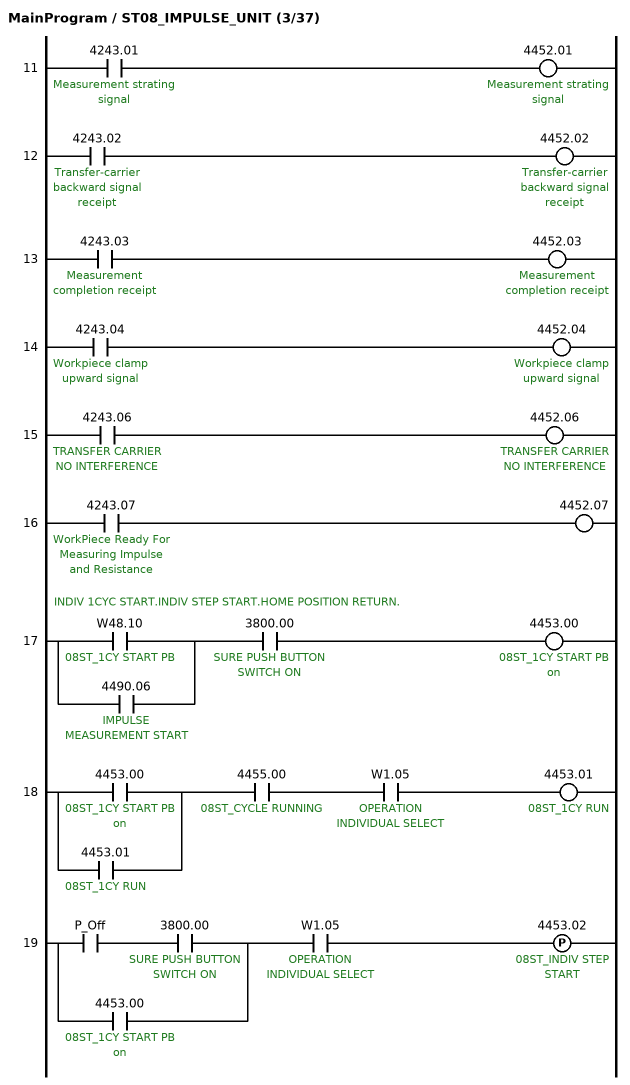
; [picture p432: MainProgram / ST08_IMPULSE_UNIT, rungs 11-19]
; rung 11
LD 4243.01  ; Measurement strating signal
OUT 4452.01  ; Measurement strating signal
; rung 12
LD 4243.02  ; Transfer-carrier backward signal receipt
OUT 4452.02  ; Transfer-carrier backward signal receipt
; rung 13
LD 4243.03  ; Measurement completion receipt
OUT 4452.03  ; Measurement completion receipt
; rung 14
LD 4243.04  ; Workpiece clamp upward signal
OUT 4452.04  ; Workpiece clamp upward signal
; rung 15
LD 4243.06  ; TRANSFER CARRIER NO INTERFERENCE
OUT 4452.06  ; TRANSFER CARRIER NO INTERFERENCE
; rung 16
LD 4243.07  ; WorkPiece Ready For Measuring Impulse and Resistance
OUT 4452.07
; rung 17: INDIV 1CYC START.INDIV STEP START.HOME POSITION RETURN.
LD W48.10  ; 08ST_1CY START PB
OR 4490.06  ; IMPULSE MEASUREMENT START
AND 3800.00  ; SURE PUSH BUTTON SWITCH ON
OUT 4453.00  ; 08ST_1CY START PB on
; rung 18
LD 4453.00  ; 08ST_1CY START PB on
OR 4453.01  ; 08ST_1CY RUN
AND 4455.00  ; 08ST_CYCLE RUNNING
AND W1.05  ; OPERATION INDIVIDUAL SELECT
OUT 4453.01  ; 08ST_1CY RUN
; rung 19
LD P_Off
AND 3800.00  ; SURE PUSH BUTTON SWITCH ON
OR 4453.00  ; 08ST_1CY START PB on
AND W1.05  ; OPERATION INDIVIDUAL SELECT
DIFU(013) 4453.02  ; 08ST_INDIV STEP START

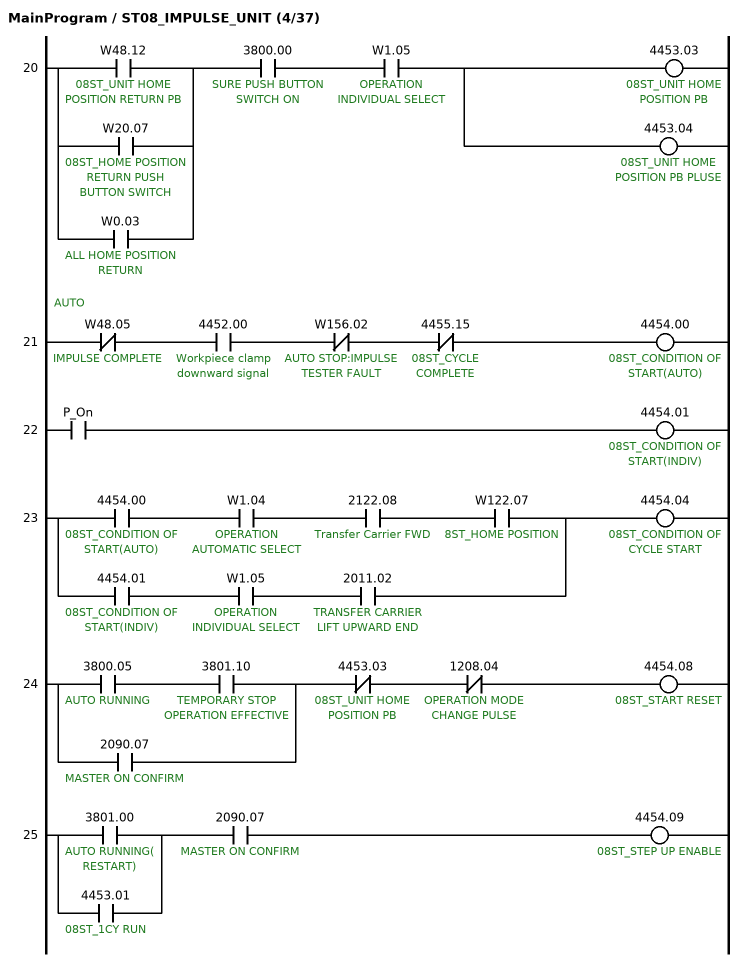
; rung 20
LD W48.12  ; 08ST_UNIT HOME POSITION RETURN PB
OR W20.07  ; 08ST_HOME POSITION RETURN PUSH BUTTON SWITCH
OR W0.03  ; ALL HOME POSITION RETURN
AND 3800.00  ; SURE PUSH BUTTON SWITCH ON
AND W1.05  ; OPERATION INDIVIDUAL SELECT
OUT 4453.03  ; 08ST_UNIT HOME POSITION PB
OUT 4453.04  ; 08ST_UNIT HOME POSITION PB PLUSE
; rung 21: AUTO
LDNOT W48.05  ; IMPULSE COMPLETE
AND 4452.00  ; Workpiece clamp downward signal
ANDNOT W156.02  ; AUTO STOP:IMPULSE TESTER FAULT
ANDNOT 4455.15  ; 08ST_CYCLE COMPLETE
OUT 4454.00  ; 08ST_CONDITION OF START(AUTO)
; rung 22
LD P_On
OUT 4454.01  ; 08ST_CONDITION OF START(INDIV)
; rung 23
LD 4454.00  ; 08ST_CONDITION OF START(AUTO)
AND W1.04  ; OPERATION AUTOMATIC SELECT
AND 2122.08  ; Transfer Carrier FWD
AND W122.07  ; 8ST_HOME POSITION
LD 4454.01  ; 08ST_CONDITION OF START(INDIV)
AND W1.05  ; OPERATION INDIVIDUAL SELECT
AND 2011.02  ; TRANSFER CARRIER LIFT UPWARD END
ORLD
OUT 4454.04  ; 08ST_CONDITION OF CYCLE START
; rung 24
LD 3800.05  ; AUTO RUNNING
AND 3801.10  ; TEMPORARY STOP OPERATION EFFECTIVE
OR 2090.07  ; MASTER ON CONFIRM
ANDNOT 4453.03  ; 08ST_UNIT HOME POSITION PB
ANDNOT 1208.04  ; OPERATION MODE CHANGE PULSE
OUT 4454.08  ; 08ST_START RESET
; rung 25
LD 3801.00  ; AUTO RUNNING(RESTART)
OR 4453.01  ; 08ST_1CY RUN
AND 2090.07  ; MASTER ON CONFIRM
OUT 4454.09  ; 08ST_STEP UP ENABLE

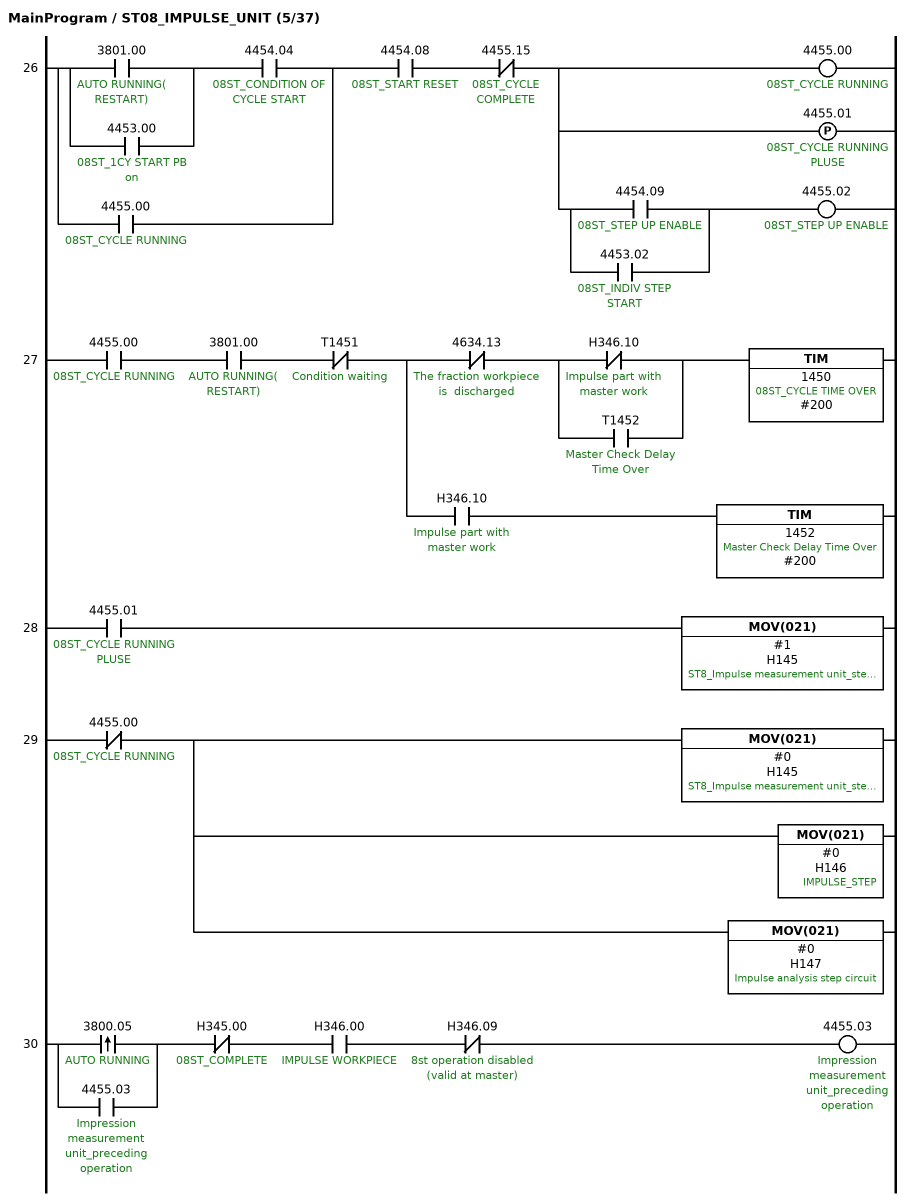
; rung 26
LD 3801.00  ; AUTO RUNNING(RESTART)
OR 4453.00  ; 08ST_1CY START PB on
AND 4454.04  ; 08ST_CONDITION OF CYCLE START
OR 4455.00  ; 08ST_CYCLE RUNNING
AND 4454.08  ; 08ST_START RESET
ANDNOT 4455.15  ; 08ST_CYCLE COMPLETE
OUT 4455.00  ; 08ST_CYCLE RUNNING
DIFU(013) 4455.01  ; 08ST_CYCLE RUNNING PLUSE
LD 4454.09  ; 08ST_STEP UP ENABLE
OR 4453.02  ; 08ST_INDIV STEP START
ANDLD
OUT 4455.02  ; 08ST_STEP UP ENABLE
; rung 27
LD 4455.00  ; 08ST_CYCLE RUNNING
AND 3801.00  ; AUTO RUNNING(RESTART)
ANDNOT T1451  ; Condition waiting
OUT TR0
ANDNOT 4634.13  ; The fraction workpiece is  discharged
LDNOT H346.10  ; Impulse part with master work
OR T1452  ; Master Check Delay Time Over
ANDLD
TIM 1450 #200  ; 08ST_CYCLE TIME OVER
LD TR0
AND H346.10  ; Impulse part with master work
TIM 1452 #200  ; Master Check Delay Time Over
; rung 28
LD 4455.01  ; 08ST_CYCLE RUNNING PLUSE
MOV(021) #1 H145  ; ST8_Impulse measurement unit_step circuit
; rung 29
LDNOT 4455.00  ; 08ST_CYCLE RUNNING
MOV(021) #0 H145  ; ST8_Impulse measurement unit_step circuit
MOV(021) #0 H146  ; IMPULSE_STEP
MOV(021) #0 H147  ; Impulse analysis step circuit
; rung 30
@LD 3800.05  ; AUTO RUNNING
OR 4455.03  ; Impression measurement unit_preceding operation
ANDNOT H345.00  ; 08ST_COMPLETE
AND H346.00  ; IMPULSE WORKPIECE
ANDNOT H346.09  ; 8st operation disabled (valid at master)
OUT 4455.03  ; Impression measurement unit_preceding operation

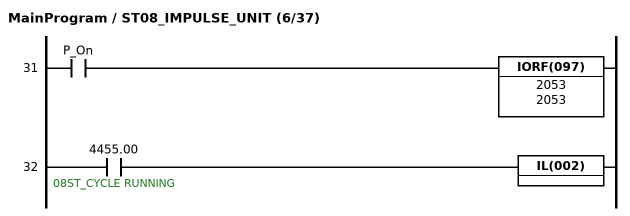
; rung 31
LD P_On
IORF(097) 2053 2053
; rung 32
LD 4455.00  ; 08ST_CYCLE RUNNING
IL(002)

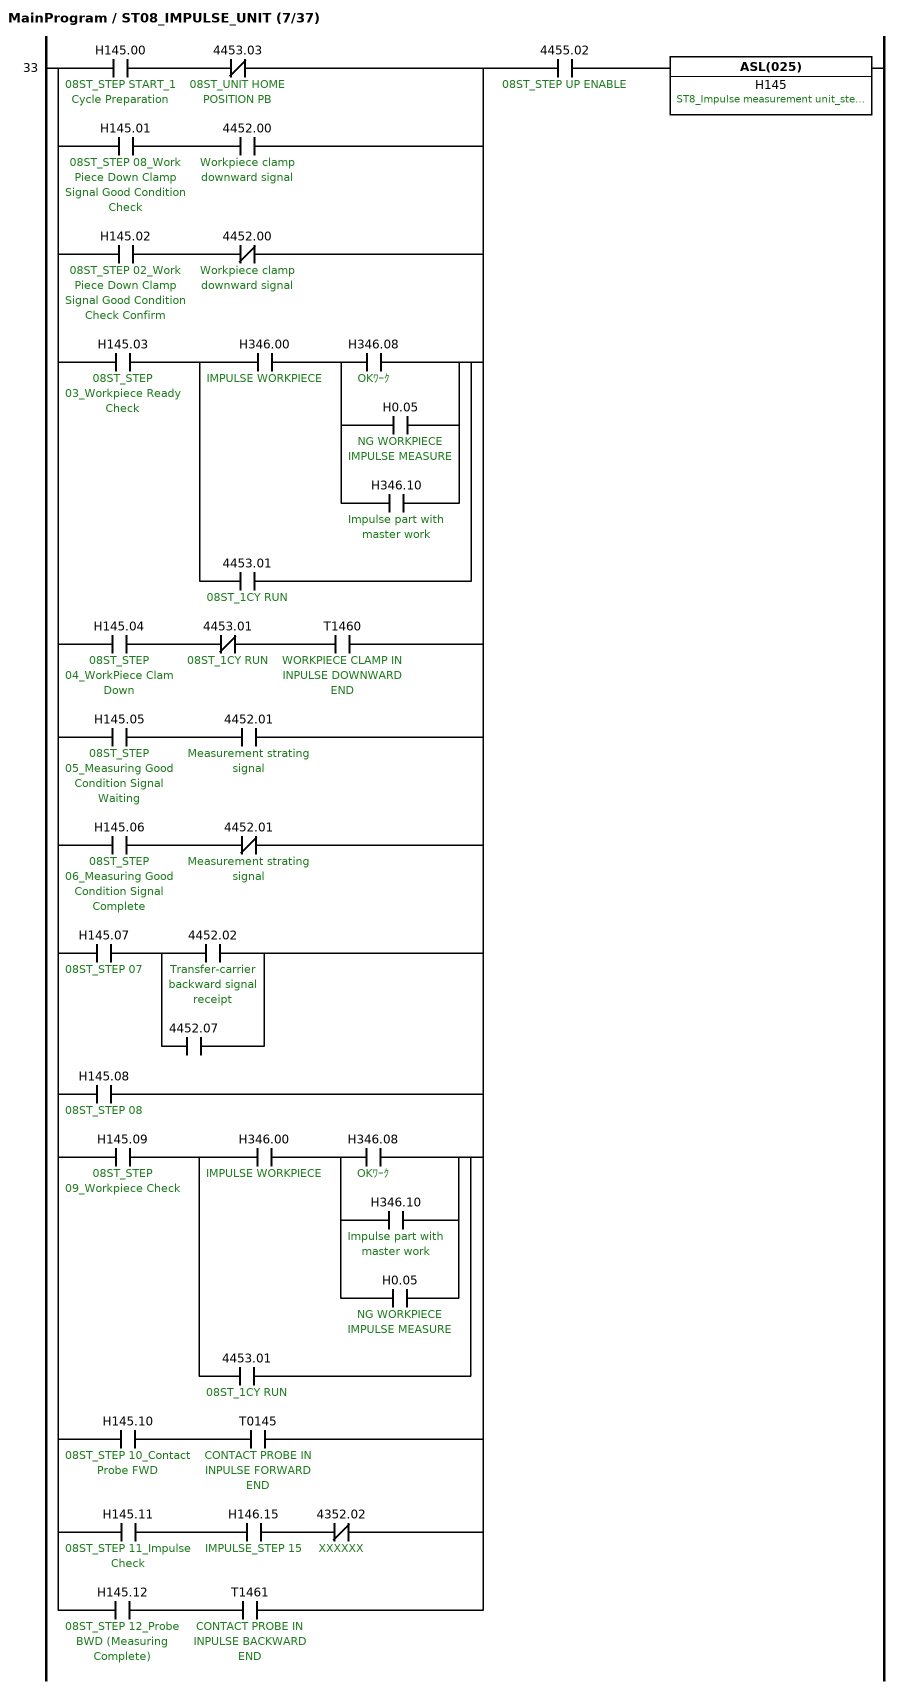
; rung 33
LD H145.00  ; 08ST_STEP START_1 Cycle Preparation
ANDNOT 4453.03  ; 08ST_UNIT HOME POSITION PB
LD H145.01  ; 08ST_STEP 08_Work Piece Down Clamp Signal Good Condition Check
AND 4452.00  ; Workpiece clamp downward signal
ORLD
LD H145.02  ; 08ST_STEP 02_Work Piece Down Clamp Signal Good Condition Check Confirm
ANDNOT 4452.00  ; Workpiece clamp downward signal
ORLD
LD H145.03  ; 08ST_STEP 03_Workpiece Ready Check
LD H346.00  ; IMPULSE WORKPIECE
LD H346.08  ; OKﾜｰｸ
OR H0.05  ; NG WORKPIECE IMPULSE MEASURE
OR H346.10  ; Impulse part with master work
ANDLD
OR 4453.01  ; 08ST_1CY RUN
ANDLD
ORLD
LD H145.04  ; 08ST_STEP 04_WorkPiece Clam Down
ANDNOT 4453.01  ; 08ST_1CY RUN
AND T1460  ; WORKPIECE CLAMP IN INPULSE DOWNWARD END
ORLD
LD H145.05  ; 08ST_STEP 05_Measuring Good Condition Signal Waiting
AND 4452.01  ; Measurement strating signal
ORLD
LD H145.06  ; 08ST_STEP 06_Measuring Good Condition Signal Complete
ANDNOT 4452.01  ; Measurement strating signal
ORLD
LD H145.07  ; 08ST_STEP 07
LD 4452.02  ; Transfer-carrier backward signal receipt
OR 4452.07
ANDLD
ORLD
OR H145.08  ; 08ST_STEP 08
LD H145.09  ; 08ST_STEP 09_Workpiece Check
LD H346.00  ; IMPULSE WORKPIECE
LD H346.08  ; OKﾜｰｸ
OR H346.10  ; Impulse part with master work
OR H0.05  ; NG WORKPIECE IMPULSE MEASURE
ANDLD
OR 4453.01  ; 08ST_1CY RUN
ANDLD
ORLD
LD H145.10  ; 08ST_STEP 10_Contact Probe FWD
AND T0145  ; CONTACT PROBE IN INPULSE FORWARD END
ORLD
LD H145.11  ; 08ST_STEP 11_Impulse Check
AND H146.15  ; IMPULSE_STEP 15
ANDNOT 4352.02  ; XXXXXX
ORLD
LD H145.12  ; 08ST_STEP 12_Probe BWD (Measuring Complete)
AND T1461  ; CONTACT PROBE IN INPULSE BACKWARD END
ORLD
AND 4455.02  ; 08ST_STEP UP ENABLE
ASL(025) H145  ; ST8_Impulse measurement unit_step circuit

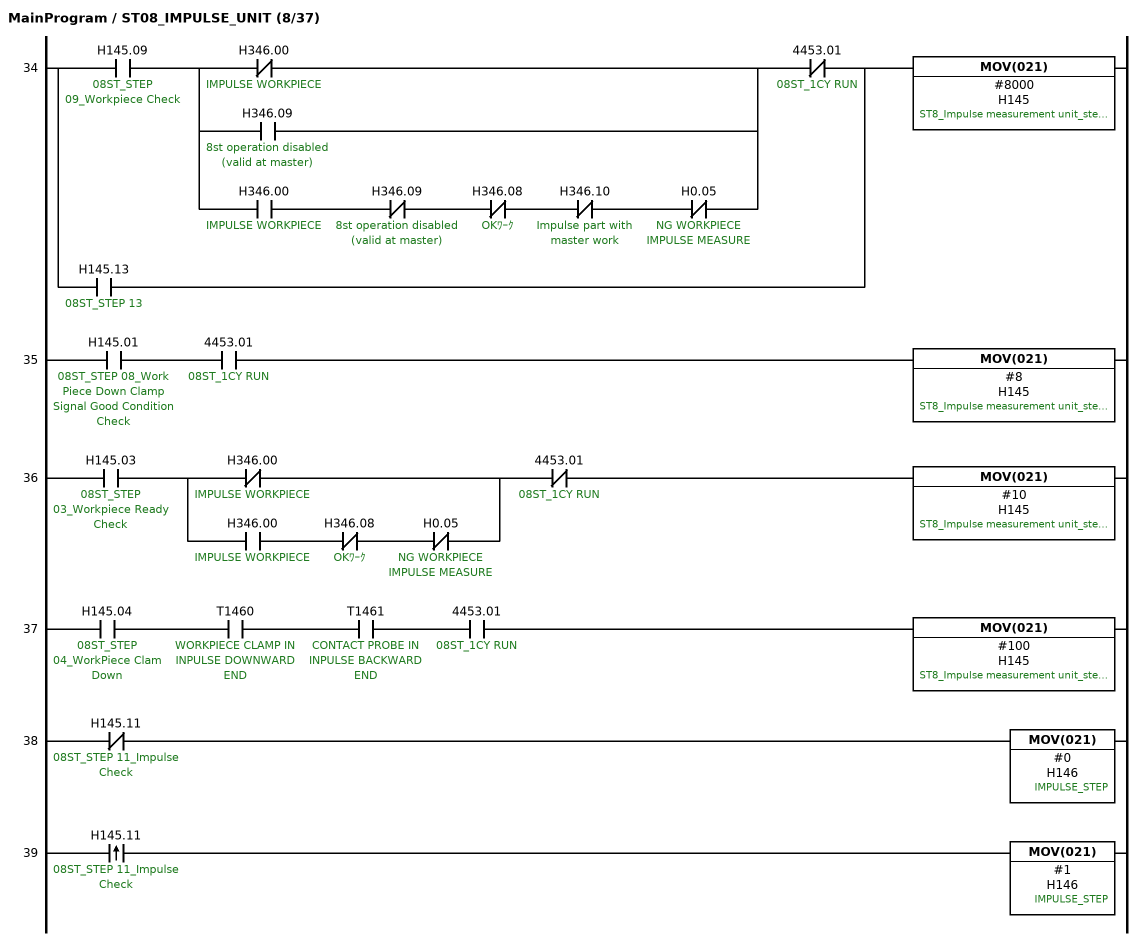
; rung 34
LD H145.09  ; 08ST_STEP 09_Workpiece Check
LDNOT H346.00  ; IMPULSE WORKPIECE
OR H346.09  ; 8st operation disabled (valid at master)
LD H346.00  ; IMPULSE WORKPIECE
ANDNOT H346.09  ; 8st operation disabled (valid at master)
ANDNOT H346.08  ; OKﾜｰｸ
ANDNOT H346.10  ; Impulse part with master work
ANDNOT H0.05  ; NG WORKPIECE IMPULSE MEASURE
ORLD
ANDLD
ANDNOT 4453.01  ; 08ST_1CY RUN
OR H145.13  ; 08ST_STEP 13
MOV(021) #8000 H145  ; ST8_Impulse measurement unit_step circuit
; rung 35
LD H145.01  ; 08ST_STEP 08_Work Piece Down Clamp Signal Good Condition Check
AND 4453.01  ; 08ST_1CY RUN
MOV(021) #8 H145  ; ST8_Impulse measurement unit_step circuit
; rung 36
LD H145.03  ; 08ST_STEP 03_Workpiece Ready Check
LDNOT H346.00  ; IMPULSE WORKPIECE
LD H346.00  ; IMPULSE WORKPIECE
ANDNOT H346.08  ; OKﾜｰｸ
ANDNOT H0.05  ; NG WORKPIECE IMPULSE MEASURE
ORLD
ANDLD
ANDNOT 4453.01  ; 08ST_1CY RUN
MOV(021) #10 H145  ; ST8_Impulse measurement unit_step circuit
; rung 37
LD H145.04  ; 08ST_STEP 04_WorkPiece Clam Down
AND T1460  ; WORKPIECE CLAMP IN INPULSE DOWNWARD END
AND T1461  ; CONTACT PROBE IN INPULSE BACKWARD END
AND 4453.01  ; 08ST_1CY RUN
MOV(021) #100 H145  ; ST8_Impulse measurement unit_step circuit
; rung 38
LDNOT H145.11  ; 08ST_STEP 11_Impulse Check
MOV(021) #0 H146  ; IMPULSE_STEP
; rung 39
@LD H145.11  ; 08ST_STEP 11_Impulse Check
MOV(021) #1 H146  ; IMPULSE_STEP

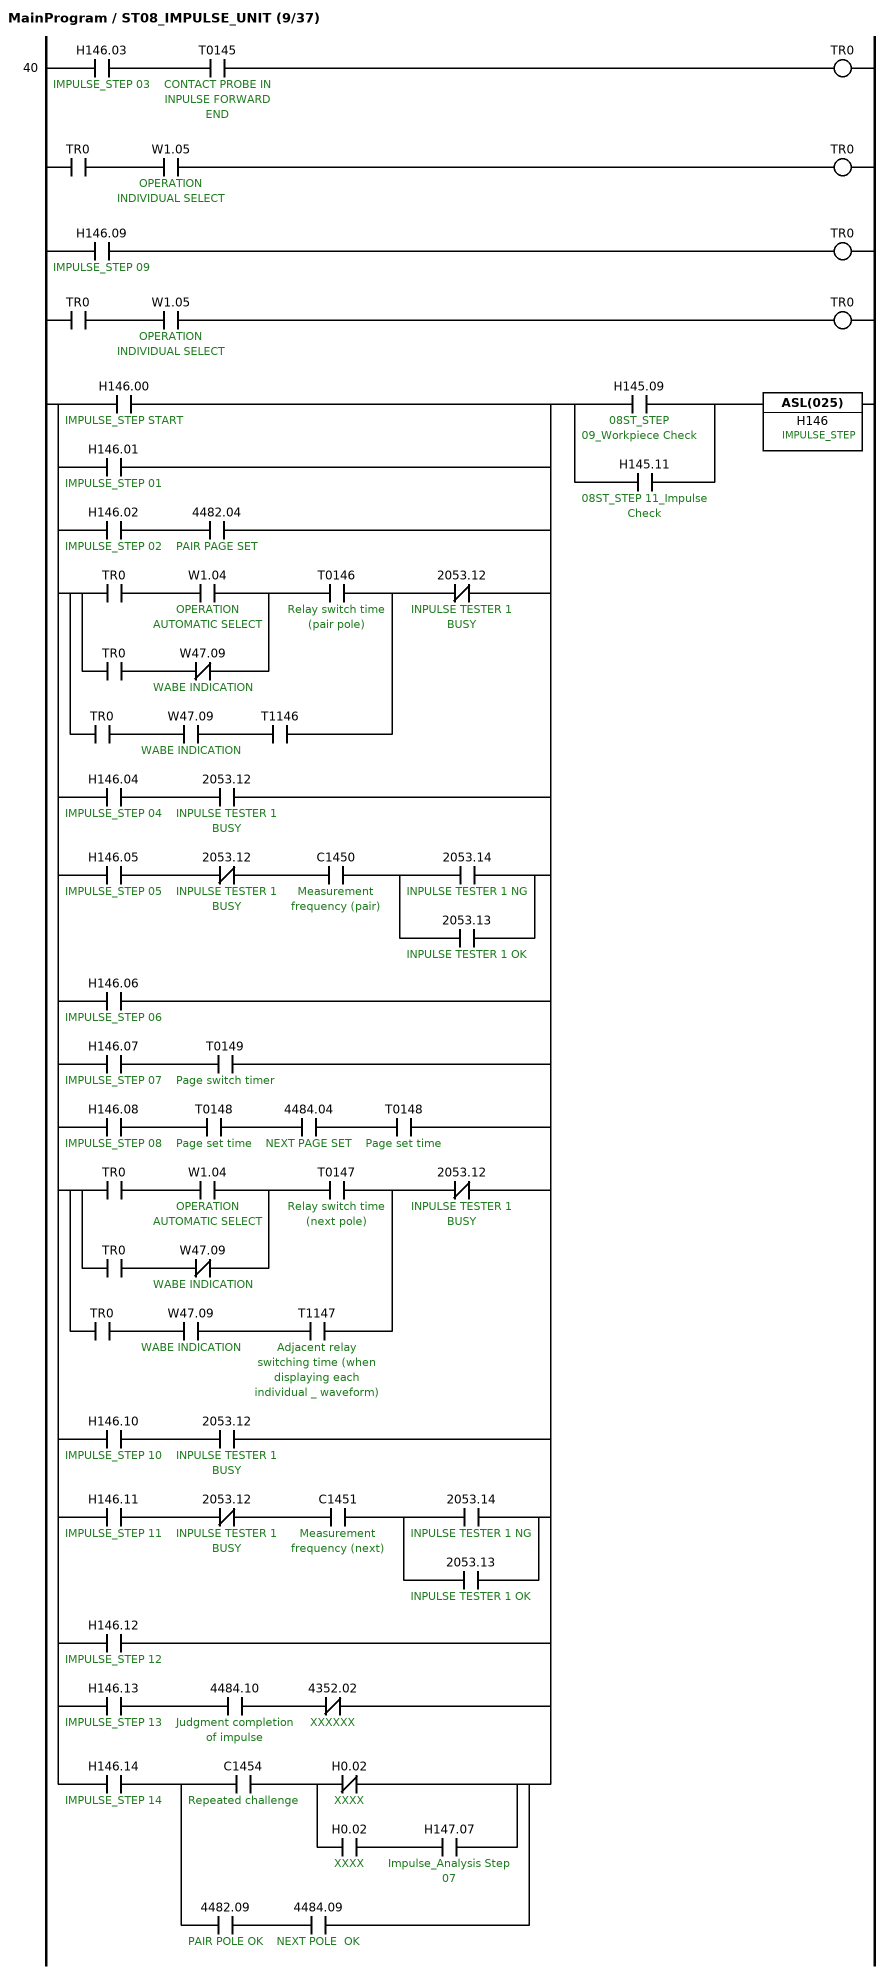
; rung 40
LD H146.00  ; IMPULSE_STEP START
OR H146.01  ; IMPULSE_STEP 01
LD H146.02  ; IMPULSE_STEP 02
AND 4482.04  ; PAIR PAGE SET
ORLD
LD H146.03  ; IMPULSE_STEP 03
AND T0145  ; CONTACT PROBE IN INPULSE FORWARD END
OUT TR0
AND W1.04  ; OPERATION AUTOMATIC SELECT
LD TR0
AND W1.05  ; OPERATION INDIVIDUAL SELECT
OUT TR0
ANDNOT W47.09  ; WABE INDICATION
ORLD
AND T0146  ; Relay switch time (pair pole)
LD TR0
AND W47.09  ; WABE INDICATION
AND T1146
ORLD
ANDNOT 2053.12  ; INPULSE TESTER 1 BUSY
ORLD
LD H146.04  ; IMPULSE_STEP 04
AND 2053.12  ; INPULSE TESTER 1 BUSY
LD H146.05  ; IMPULSE_STEP 05
ANDNOT 2053.12  ; INPULSE TESTER 1 BUSY
AND C1450  ; Measurement frequency (pair)
LD 2053.14  ; INPULSE TESTER 1 NG
OR 2053.13  ; INPULSE TESTER 1 OK
ANDLD
ORLD
OR H146.06  ; IMPULSE_STEP 06
LD H146.07  ; IMPULSE_STEP 07
AND T0149  ; Page switch timer
ORLD
LD H146.08  ; IMPULSE_STEP 08
AND T0148  ; Page set time
AND 4484.04  ; NEXT PAGE SET
AND T0148  ; Page set time
ORLD
ORLD
LD H146.09  ; IMPULSE_STEP 09
OUT TR0
AND W1.04  ; OPERATION AUTOMATIC SELECT
LD TR0
AND W1.05  ; OPERATION INDIVIDUAL SELECT
OUT TR0
ANDNOT W47.09  ; WABE INDICATION
ORLD
AND T0147  ; Relay switch time (next pole)
LD TR0
AND W47.09  ; WABE INDICATION
AND T1147  ; Adjacent relay switching time (when displaying each individual _ waveform)
ORLD
ANDNOT 2053.12  ; INPULSE TESTER 1 BUSY
ORLD
LD H146.10  ; IMPULSE_STEP 10
AND 2053.12  ; INPULSE TESTER 1 BUSY
LD H146.11  ; IMPULSE_STEP 11
ANDNOT 2053.12  ; INPULSE TESTER 1 BUSY
AND C1451  ; Measurement frequency (next)
LD 2053.14  ; INPULSE TESTER 1 NG
OR 2053.13  ; INPULSE TESTER 1 OK
ANDLD
ORLD
OR H146.12  ; IMPULSE_STEP 12
LD H146.13  ; IMPULSE_STEP 13
AND 4484.10  ; Judgment completion of impulse
ANDNOT 4352.02  ; XXXXXX
ORLD
LD H146.14  ; IMPULSE_STEP 14
LD C1454  ; Repeated challenge
LDNOT H0.02  ; XXXX
LD H0.02  ; XXXX
AND H147.07  ; Impulse_Analysis Step 07
ORLD
ANDLD
LD 4482.09  ; PAIR POLE OK
AND 4484.09  ; NEXT POLE  OK
ORLD
ANDLD
ORLD
ORLD
LD H145.09  ; 08ST_STEP 09_Workpiece Check
OR H145.11  ; 08ST_STEP 11_Impulse Check
ANDLD
ASL(025) H146  ; IMPULSE_STEP

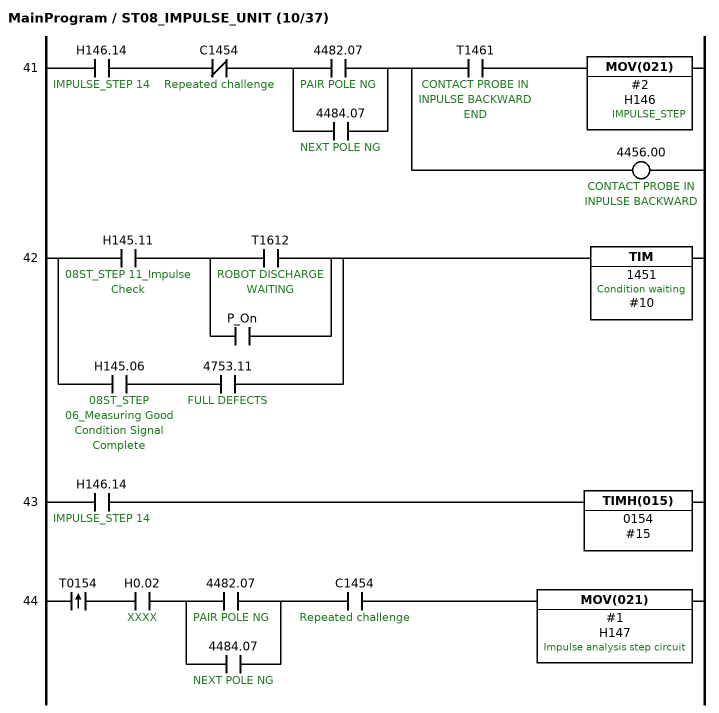
; rung 41
LD H146.14  ; IMPULSE_STEP 14
ANDNOT C1454  ; Repeated challenge
LD 4482.07  ; PAIR POLE NG
OR 4484.07  ; NEXT POLE NG
ANDLD
OUT TR0
AND T1461  ; CONTACT PROBE IN INPULSE BACKWARD END
MOV(021) #2 H146  ; IMPULSE_STEP
LD TR0
OUT 4456.00  ; CONTACT PROBE IN INPULSE BACKWARD
; rung 42
LD H145.11  ; 08ST_STEP 11_Impulse Check
LD T1612  ; ROBOT DISCHARGE WAITING
OR P_On
ANDLD
LD H145.06  ; 08ST_STEP 06_Measuring Good Condition Signal Complete
AND 4753.11  ; FULL DEFECTS
ORLD
TIM 1451 #10  ; Condition waiting  // from 50 => 10
; rung 43
LD H146.14  ; IMPULSE_STEP 14
TIMH(015) 0154 #15
; rung 44
@LD T0154
AND H0.02  ; XXXX
LD 4482.07  ; PAIR POLE NG
OR 4484.07  ; NEXT POLE NG
ANDLD
AND C1454  ; Repeated challenge
MOV(021) #1 H147  ; Impulse analysis step circuit

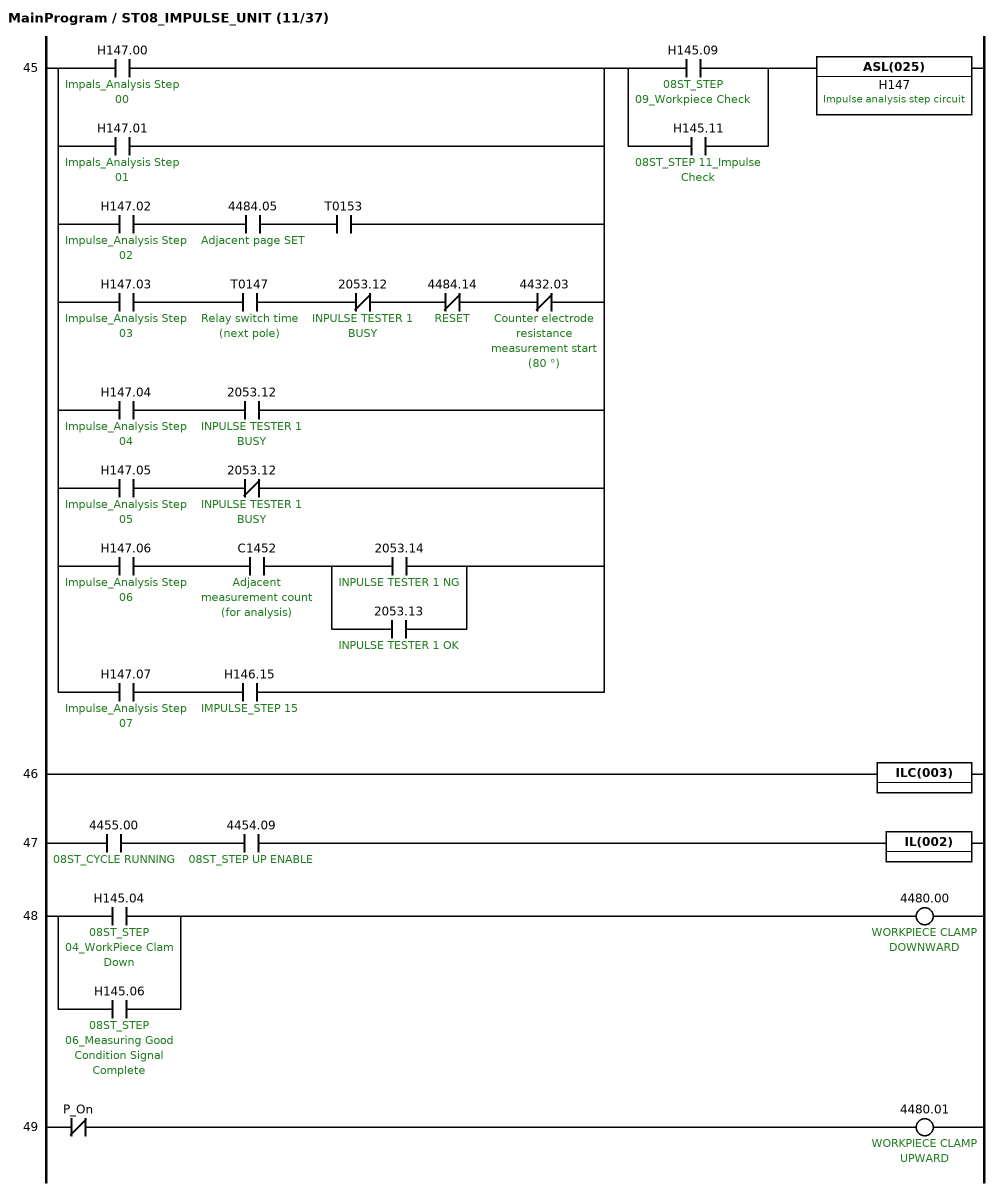
; rung 45
LD H147.00  ; Impals_Analysis Step 00
OR H147.01  ; Impals_Analysis Step 01
LD H147.02  ; Impulse_Analysis Step 02
AND 4484.05  ; Adjacent page SET
AND T0153
ORLD
LD H147.03  ; Impulse_Analysis Step 03
AND T0147  ; Relay switch time (next pole)
ANDNOT 2053.12  ; INPULSE TESTER 1 BUSY
ANDNOT 4484.14  ; RESET
ANDNOT 4432.03  ; Counter electrode resistance measurement start (80 °)
ORLD
LD H147.04  ; Impulse_Analysis Step 04
AND 2053.12  ; INPULSE TESTER 1 BUSY
ORLD
LD H147.05  ; Impulse_Analysis Step 05
ANDNOT 2053.12  ; INPULSE TESTER 1 BUSY
ORLD
LD H147.06  ; Impulse_Analysis Step 06
AND C1452  ; Adjacent measurement count (for analysis)
LD 2053.14  ; INPULSE TESTER 1 NG
OR 2053.13  ; INPULSE TESTER 1 OK
ANDLD
ORLD
LD H147.07  ; Impulse_Analysis Step 07
AND H146.15  ; IMPULSE_STEP 15
ORLD
LD H145.09  ; 08ST_STEP 09_Workpiece Check
OR H145.11  ; 08ST_STEP 11_Impulse Check
ANDLD
ASL(025) H147  ; Impulse analysis step circuit
; rung 46
ILC(003)
; rung 47
LD 4455.00  ; 08ST_CYCLE RUNNING
AND 4454.09  ; 08ST_STEP UP ENABLE
IL(002)
; rung 48
LD H145.04  ; 08ST_STEP 04_WorkPiece Clam Down
OR H145.06  ; 08ST_STEP 06_Measuring Good Condition Signal Complete
OUT 4480.00  ; WORKPIECE CLAMP DOWNWARD
; rung 49
LDNOT P_On
OUT 4480.01  ; WORKPIECE CLAMP UPWARD

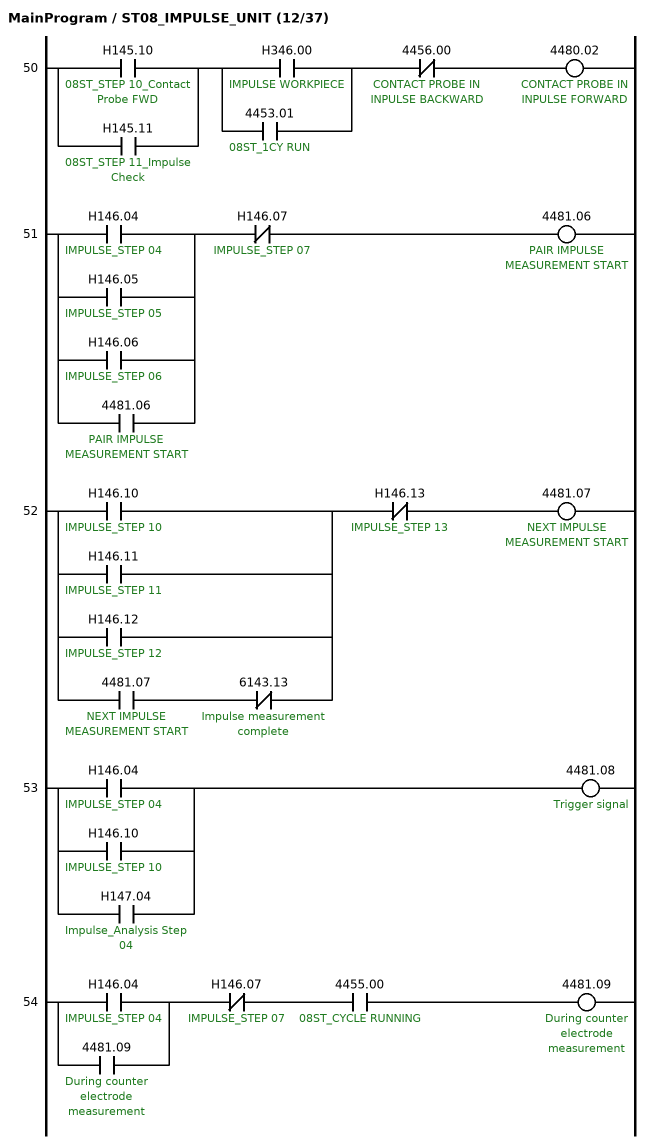
; rung 50
LD H145.10  ; 08ST_STEP 10_Contact Probe FWD
OR H145.11  ; 08ST_STEP 11_Impulse Check
LD H346.00  ; IMPULSE WORKPIECE
OR 4453.01  ; 08ST_1CY RUN
ANDLD
ANDNOT 4456.00  ; CONTACT PROBE IN INPULSE BACKWARD
OUT 4480.02  ; CONTACT PROBE IN INPULSE FORWARD
; rung 51
LD H146.04  ; IMPULSE_STEP 04
OR H146.05  ; IMPULSE_STEP 05
LD H146.06  ; IMPULSE_STEP 06
OR 4481.06  ; PAIR IMPULSE MEASUREMENT START
ORLD
ANDNOT H146.07  ; IMPULSE_STEP 07
OUT 4481.06  ; PAIR IMPULSE MEASUREMENT START
; rung 52
LD H146.10  ; IMPULSE_STEP 10
OR H146.11  ; IMPULSE_STEP 11
OR H146.12  ; IMPULSE_STEP 12
LD 4481.07  ; NEXT IMPULSE MEASUREMENT START
ANDNOT 6143.13  ; Impulse measurement complete
ORLD
ANDNOT H146.13  ; IMPULSE_STEP 13
OUT 4481.07  ; NEXT IMPULSE MEASUREMENT START
; rung 53
LD H146.04  ; IMPULSE_STEP 04
OR H146.10  ; IMPULSE_STEP 10
OR H147.04  ; Impulse_Analysis Step 04
OUT 4481.08  ; Trigger signal
; rung 54
LD H146.04  ; IMPULSE_STEP 04
OR 4481.09  ; During counter electrode measurement
ANDNOT H146.07  ; IMPULSE_STEP 07
AND 4455.00  ; 08ST_CYCLE RUNNING
OUT 4481.09  ; During counter electrode measurement

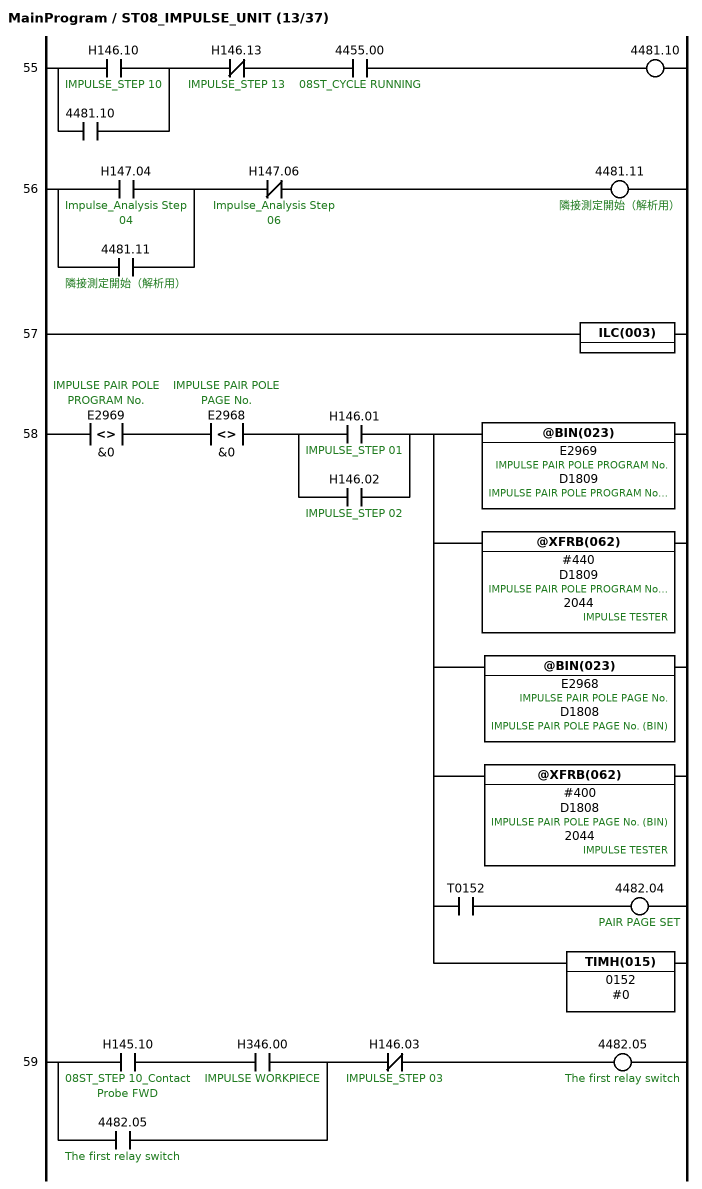
; rung 55
LD H146.10  ; IMPULSE_STEP 10
OR 4481.10
ANDNOT H146.13  ; IMPULSE_STEP 13
AND 4455.00  ; 08ST_CYCLE RUNNING
OUT 4481.10
; rung 56
LD H147.04  ; Impulse_Analysis Step 04
OR 4481.11  ; 隣接測定開始（解析用）
ANDNOT H147.06  ; Impulse_Analysis Step 06
OUT 4481.11  ; 隣接測定開始（解析用）
; rung 57
ILC(003)
; rung 58
LD<>(305) E2969 &0  ; IMPULSE PAIR POLE PROGRAM No.
AND<>(305) E2968 &0  ; IMPULSE PAIR POLE PAGE No.
LD H146.01  ; IMPULSE_STEP 01
OR H146.02  ; IMPULSE_STEP 02
ANDLD
OUT TR0
@BIN(023) E2969 D1809  ; IMPULSE PAIR POLE PROGRAM No., IMPULSE PAIR POLE PROGRAM No. (BIN)
@XFRB(062) #440 D1809 2044  ; IMPULSE PAIR POLE PROGRAM No. (BIN), IMPULSE TESTER
@BIN(023) E2968 D1808  ; IMPULSE PAIR POLE PAGE No., IMPULSE PAIR POLE PAGE No. (BIN)
@XFRB(062) #400 D1808 2044  ; IMPULSE PAIR POLE PAGE No. (BIN), IMPULSE TESTER
AND T0152
OUT 4482.04  ; PAIR PAGE SET
LD TR0
TIMH(015) 0152 #0
; rung 59
LD H145.10  ; 08ST_STEP 10_Contact Probe FWD
AND H346.00  ; IMPULSE WORKPIECE
OR 4482.05  ; The first relay switch
ANDNOT H146.03  ; IMPULSE_STEP 03
OUT 4482.05  ; The first relay switch

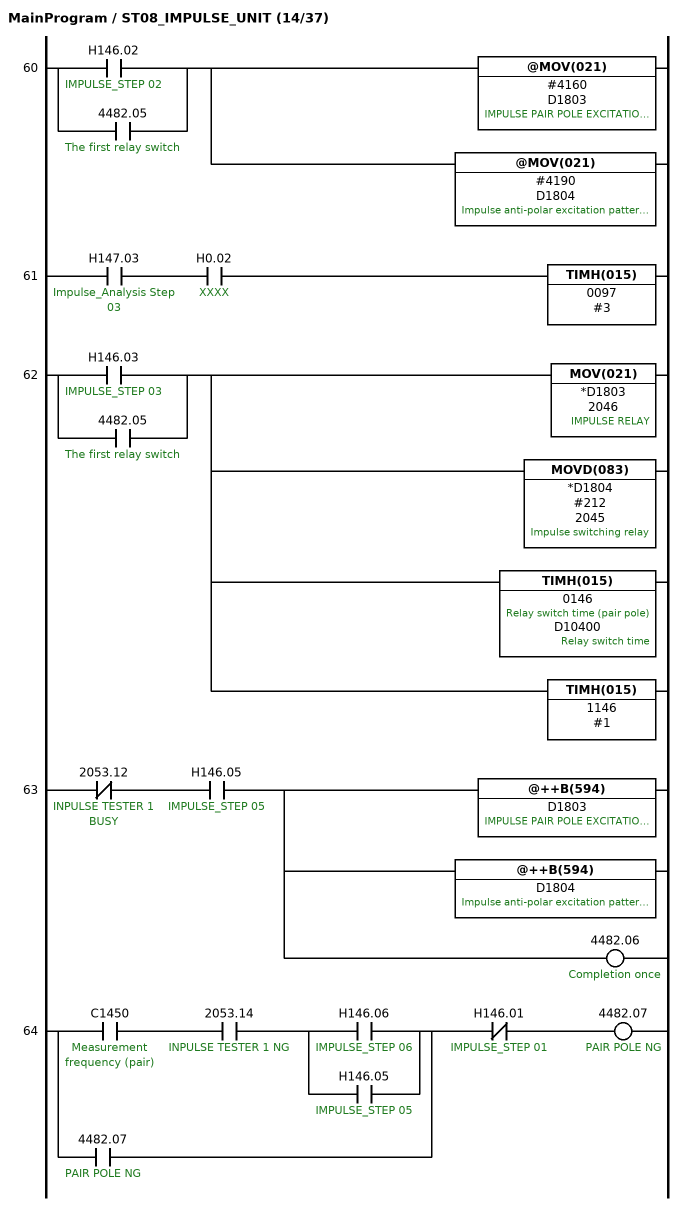
; rung 60
LD H146.02  ; IMPULSE_STEP 02
OR 4482.05  ; The first relay switch
@MOV(021) #4160 D1803  ; IMPULSE PAIR POLE EXCITATION PATTERN DM STORING
@MOV(021) #4190 D1804  ; Impulse anti-polar excitation pattern storage
; rung 61
LD H147.03  ; Impulse_Analysis Step 03
AND H0.02  ; XXXX
TIMH(015) 0097 #3
; rung 62
LD H146.03  ; IMPULSE_STEP 03
OR 4482.05  ; The first relay switch
MOV(021) *D1803 2046  ; IMPULSE RELAY
MOVD(083) *D1804 #212 2045  ; Impulse switching relay
TIMH(015) 0146 D10400  ; Relay switch time, Relay switch time (pair pole)
TIMH(015) 1146 #1
; rung 63
LDNOT 2053.12  ; INPULSE TESTER 1 BUSY
AND H146.05  ; IMPULSE_STEP 05
@++B(594) D1803  ; IMPULSE PAIR POLE EXCITATION PATTERN DM STORING
@++B(594) D1804  ; Impulse anti-polar excitation pattern storage
OUT 4482.06  ; Completion once
; rung 64
LD C1450  ; Measurement frequency (pair)
AND 2053.14  ; INPULSE TESTER 1 NG
LD H146.06  ; IMPULSE_STEP 06
OR H146.05  ; IMPULSE_STEP 05
ANDLD
OR 4482.07  ; PAIR POLE NG
ANDNOT H146.01  ; IMPULSE_STEP 01
OUT 4482.07  ; PAIR POLE NG

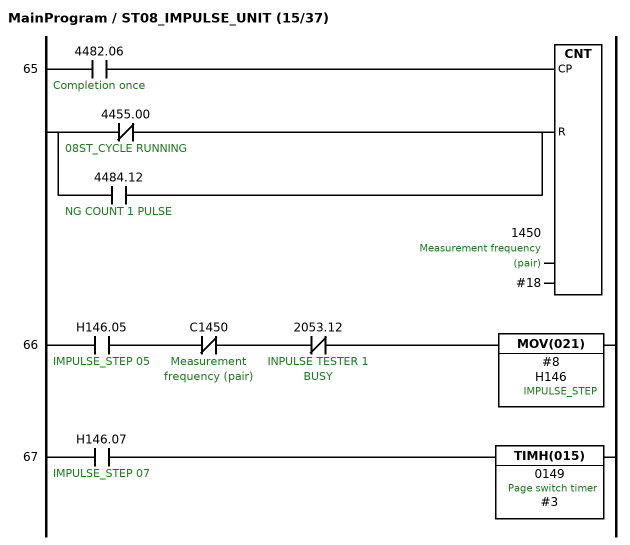
; rung 65
LD 4482.06  ; Completion once
LDNOT 4455.00  ; 08ST_CYCLE RUNNING
OR 4484.12  ; NG COUNT 1 PULSE
CNT 1450 #18  ; Measurement frequency (pair)  // 6　=>　18
; rung 66
LD H146.05  ; IMPULSE_STEP 05
ANDNOT C1450  ; Measurement frequency (pair)
ANDNOT 2053.12  ; INPULSE TESTER 1 BUSY
MOV(021) #8 H146  ; IMPULSE_STEP
; rung 67
LD H146.07  ; IMPULSE_STEP 07
TIMH(015) 0149 #3  ; Page switch timer  // 10　=>　3

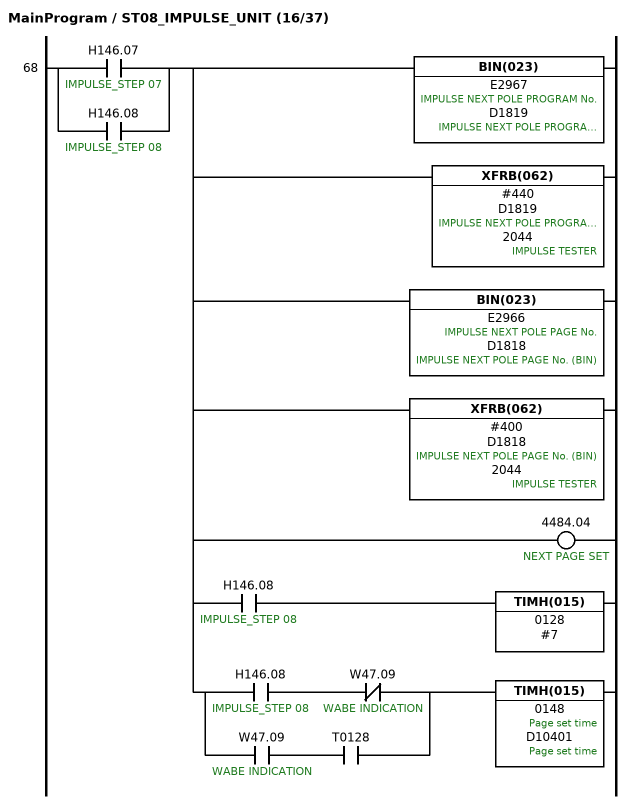
; rung 68
LD H146.07  ; IMPULSE_STEP 07
OR H146.08  ; IMPULSE_STEP 08
OUT TR0
BIN(023) E2967 D1819  ; IMPULSE NEXT POLE PROGRAM No., IMPULSE NEXT POLE PROGRAM No.(BIN)
XFRB(062) #440 D1819 2044  ; IMPULSE NEXT POLE PROGRAM No.(BIN), IMPULSE TESTER
BIN(023) E2966 D1818  ; IMPULSE NEXT POLE PAGE No., IMPULSE NEXT POLE PAGE No. (BIN)
XFRB(062) #400 D1818 2044  ; IMPULSE NEXT POLE PAGE No. (BIN), IMPULSE TESTER
OUT 4484.04  ; NEXT PAGE SET
AND H146.08  ; IMPULSE_STEP 08
TIMH(015) 0128 #7
LD TR0
LD H146.08  ; IMPULSE_STEP 08
ANDNOT W47.09  ; WABE INDICATION
LD W47.09  ; WABE INDICATION
AND T0128
ORLD
ANDLD
TIMH(015) 0148 D10401  ; Page set time

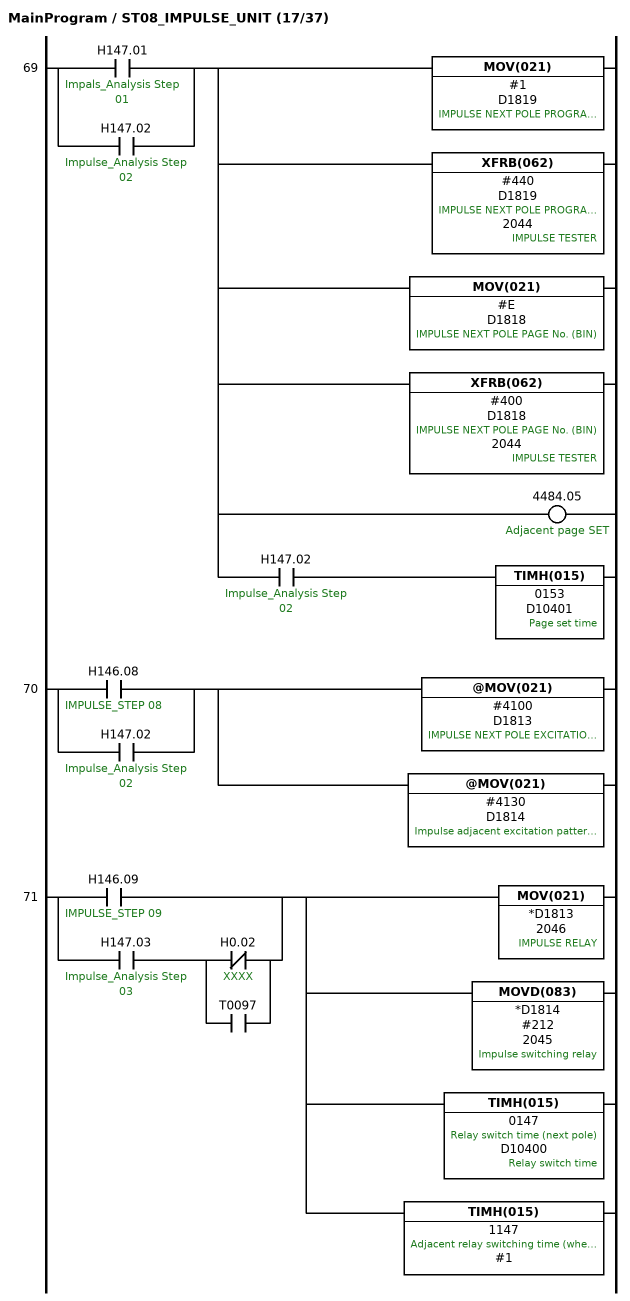
; rung 69
LD H147.01  ; Impals_Analysis Step 01
OR H147.02  ; Impulse_Analysis Step 02
MOV(021) #1 D1819  ; IMPULSE NEXT POLE PROGRAM No.(BIN)
XFRB(062) #440 D1819 2044  ; IMPULSE NEXT POLE PROGRAM No.(BIN), IMPULSE TESTER
MOV(021) #E D1818  ; IMPULSE NEXT POLE PAGE No. (BIN)
XFRB(062) #400 D1818 2044  ; IMPULSE NEXT POLE PAGE No. (BIN), IMPULSE TESTER
OUT 4484.05  ; Adjacent page SET
AND H147.02  ; Impulse_Analysis Step 02
TIMH(015) 0153 D10401  ; Page set time
; rung 70
LD H146.08  ; IMPULSE_STEP 08
OR H147.02  ; Impulse_Analysis Step 02
@MOV(021) #4100 D1813  ; IMPULSE NEXT POLE EXCITATION PATTERN DM STORING
@MOV(021) #4130 D1814  ; Impulse adjacent excitation pattern storage
; rung 71
LD H146.09  ; IMPULSE_STEP 09
LD H147.03  ; Impulse_Analysis Step 03
LDNOT H0.02  ; XXXX
OR T0097
ANDLD
ORLD
MOV(021) *D1813 2046  ; IMPULSE RELAY
MOVD(083) *D1814 #212 2045  ; Impulse switching relay
TIMH(015) 0147 D10400  ; Relay switch time, Relay switch time (next pole)
TIMH(015) 1147 #1  ; Adjacent relay switching time (when displaying each individual _ waveform)

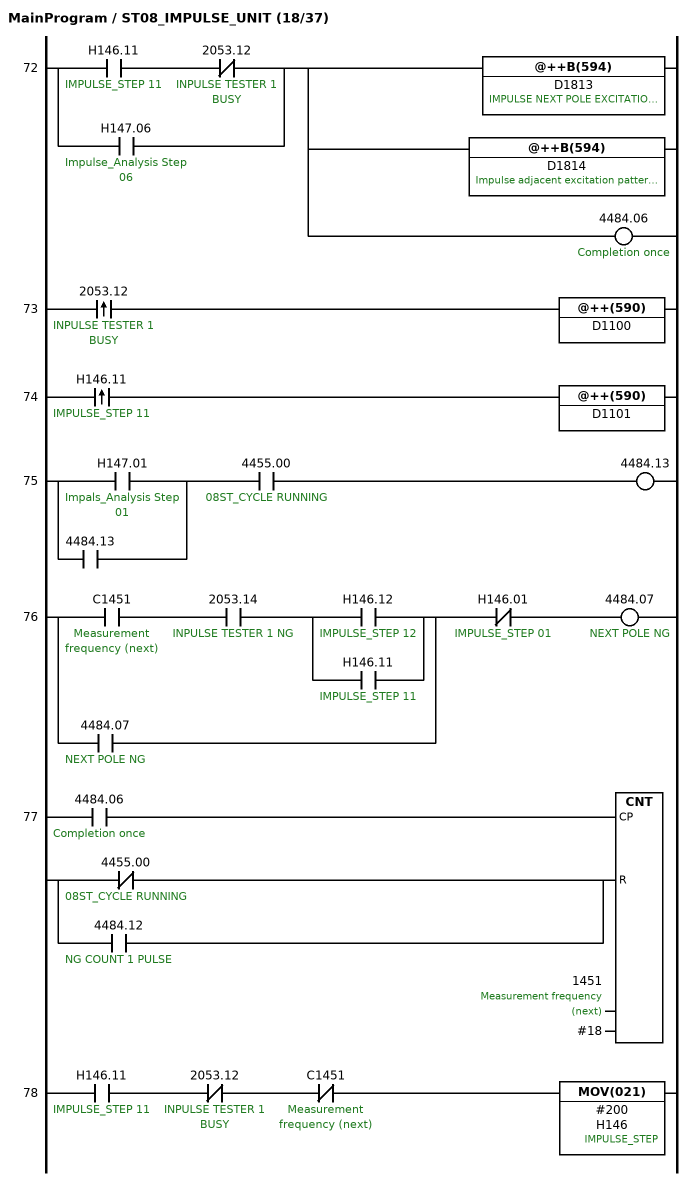
; rung 72
LD H146.11  ; IMPULSE_STEP 11
ANDNOT 2053.12  ; INPULSE TESTER 1 BUSY
OR H147.06  ; Impulse_Analysis Step 06
@++B(594) D1813  ; IMPULSE NEXT POLE EXCITATION PATTERN DM STORING
@++B(594) D1814  ; Impulse adjacent excitation pattern storage
OUT 4484.06  ; Completion once
; rung 73
@LD 2053.12  ; INPULSE TESTER 1 BUSY
@++(590) D1100
; rung 74
@LD H146.11  ; IMPULSE_STEP 11
@++(590) D1101
; rung 75
LD H147.01  ; Impals_Analysis Step 01
OR 4484.13
AND 4455.00  ; 08ST_CYCLE RUNNING
OUT 4484.13
; rung 76
LD C1451  ; Measurement frequency (next)
AND 2053.14  ; INPULSE TESTER 1 NG
LD H146.12  ; IMPULSE_STEP 12
OR H146.11  ; IMPULSE_STEP 11
ANDLD
OR 4484.07  ; NEXT POLE NG
ANDNOT H146.01  ; IMPULSE_STEP 01
OUT 4484.07  ; NEXT POLE NG
; rung 77
LD 4484.06  ; Completion once
LDNOT 4455.00  ; 08ST_CYCLE RUNNING
OR 4484.12  ; NG COUNT 1 PULSE
CNT 1451 #18  ; Measurement frequency (next)  // 12　　＝>　18
; rung 78
LD H146.11  ; IMPULSE_STEP 11
ANDNOT 2053.12  ; INPULSE TESTER 1 BUSY
ANDNOT C1451  ; Measurement frequency (next)
MOV(021) #200 H146  ; IMPULSE_STEP

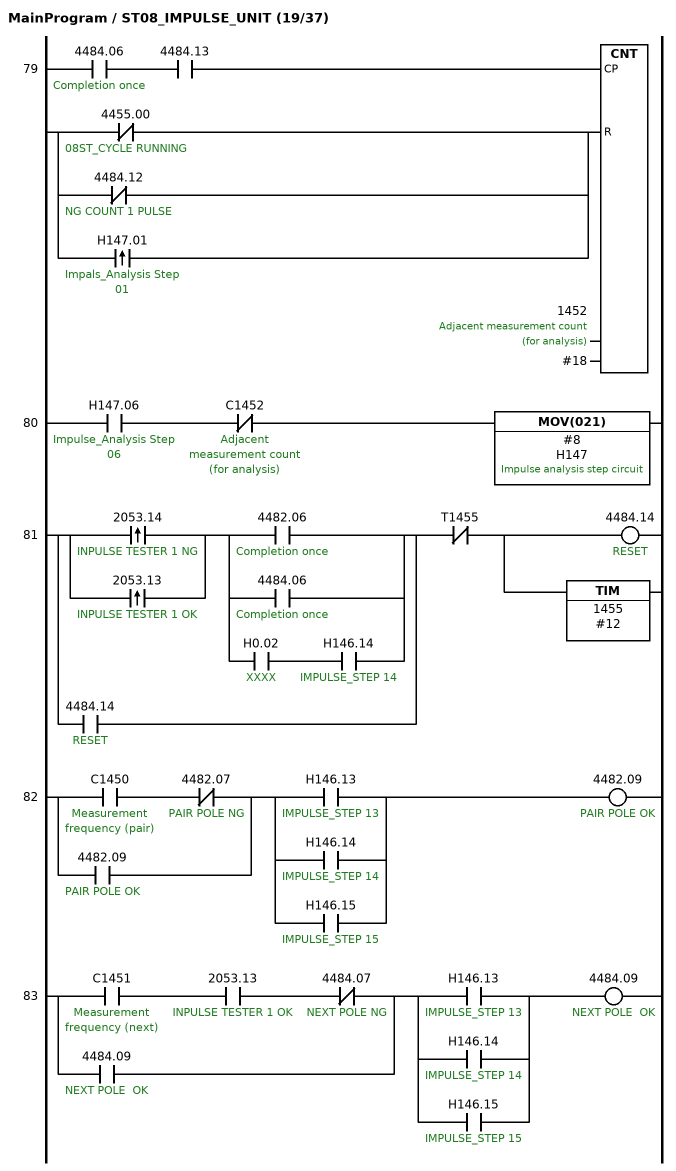
; rung 79
LD 4484.06  ; Completion once
AND 4484.13
LDNOT 4455.00  ; 08ST_CYCLE RUNNING
ORNOT 4484.12  ; NG COUNT 1 PULSE
@OR H147.01  ; Impals_Analysis Step 01
CNT 1452 #18  ; Adjacent measurement count (for analysis)
; rung 80
LD H147.06  ; Impulse_Analysis Step 06
ANDNOT C1452  ; Adjacent measurement count (for analysis)
MOV(021) #8 H147  ; Impulse analysis step circuit
; rung 81
@LD 2053.14  ; INPULSE TESTER 1 NG
@OR 2053.13  ; INPULSE TESTER 1 OK
LD 4482.06  ; Completion once
OR 4484.06  ; Completion once
LD H0.02  ; XXXX
AND H146.14  ; IMPULSE_STEP 14
ORLD
ANDLD
OR 4484.14  ; RESET
ANDNOT T1455
OUT 4484.14  ; RESET
TIM 1455 #12  // 1=>12
; rung 82
LD C1450  ; Measurement frequency (pair)
ANDNOT 4482.07  ; PAIR POLE NG
OR 4482.09  ; PAIR POLE OK
LD H146.13  ; IMPULSE_STEP 13
OR H146.14  ; IMPULSE_STEP 14
OR H146.15  ; IMPULSE_STEP 15
ANDLD
OUT 4482.09  ; PAIR POLE OK
; rung 83
LD C1451  ; Measurement frequency (next)
AND 2053.13  ; INPULSE TESTER 1 OK
ANDNOT 4484.07  ; NEXT POLE NG
OR 4484.09  ; NEXT POLE  OK
LD H146.13  ; IMPULSE_STEP 13
OR H146.14  ; IMPULSE_STEP 14
OR H146.15  ; IMPULSE_STEP 15
ANDLD
OUT 4484.09  ; NEXT POLE  OK

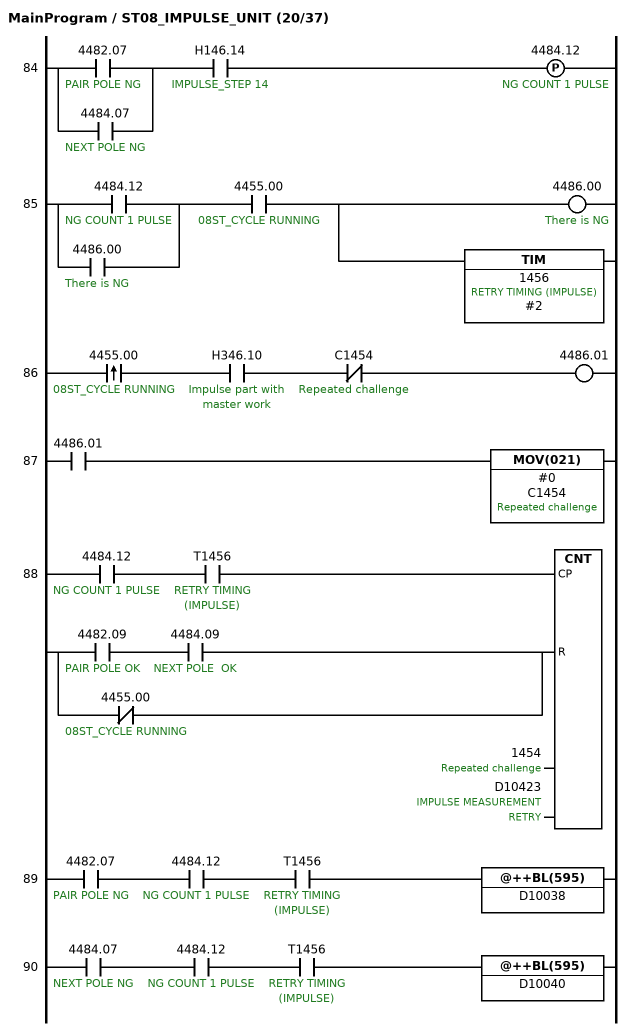
; rung 84
LD 4482.07  ; PAIR POLE NG
OR 4484.07  ; NEXT POLE NG
AND H146.14  ; IMPULSE_STEP 14
DIFU(013) 4484.12  ; NG COUNT 1 PULSE
; rung 85
LD 4484.12  ; NG COUNT 1 PULSE
OR 4486.00  ; There is NG
AND 4455.00  ; 08ST_CYCLE RUNNING
OUT 4486.00  ; There is NG
TIM 1456 #2  ; RETRY TIMING (IMPULSE)
; rung 86
@LD 4455.00  ; 08ST_CYCLE RUNNING
AND H346.10  ; Impulse part with master work
ANDNOT C1454  ; Repeated challenge
OUT 4486.01
; rung 87
LD 4486.01
MOV(021) #0 C1454  ; Repeated challenge
; rung 88
LD 4484.12  ; NG COUNT 1 PULSE
AND T1456  ; RETRY TIMING (IMPULSE)
LD 4482.09  ; PAIR POLE OK
AND 4484.09  ; NEXT POLE  OK
ORNOT 4455.00  ; 08ST_CYCLE RUNNING
CNT 1454 D10423  ; IMPULSE MEASUREMENT RETRY, Repeated challenge
; rung 89
LD 4482.07  ; PAIR POLE NG
AND 4484.12  ; NG COUNT 1 PULSE
AND T1456  ; RETRY TIMING (IMPULSE)
@++BL(595) D10038
; rung 90
LD 4484.07  ; NEXT POLE NG
AND 4484.12  ; NG COUNT 1 PULSE
AND T1456  ; RETRY TIMING (IMPULSE)
@++BL(595) D10040

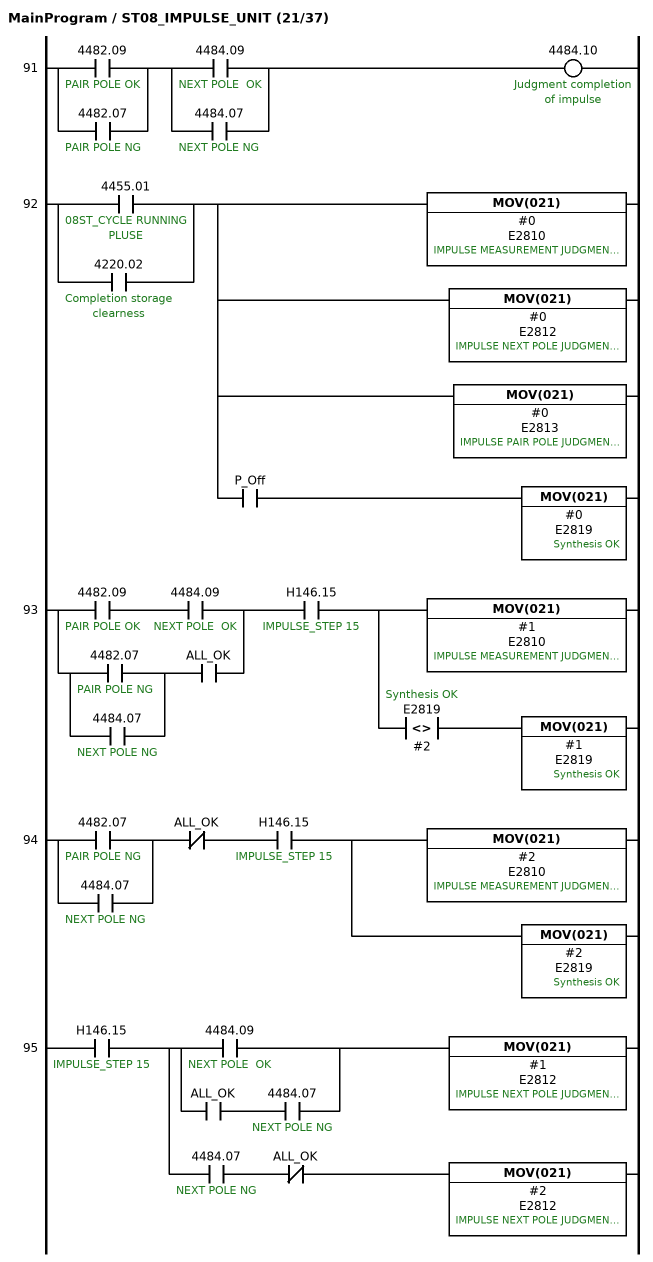
; rung 91
LD 4482.09  ; PAIR POLE OK
OR 4482.07  ; PAIR POLE NG
LD 4484.09  ; NEXT POLE  OK
OR 4484.07  ; NEXT POLE NG
ANDLD
OUT 4484.10  ; Judgment completion of impulse
; rung 92
LD 4455.01  ; 08ST_CYCLE RUNNING PLUSE
OR 4220.02  ; Completion storage clearness
MOV(021) #0 E2810  ; IMPULSE MEASUREMENT JUDGMENT RESULT (1:OK,2:NG)
MOV(021) #0 E2812  ; IMPULSE NEXT POLE JUDGMENT RESULT (1:OK,2:NG)
MOV(021) #0 E2813  ; IMPULSE PAIR POLE JUDGMENT RESULT (1:OK,2:NG)
AND P_Off
MOV(021) #0 E2819  ; Synthesis OK
; rung 93
LD 4482.09  ; PAIR POLE OK
AND 4484.09  ; NEXT POLE  OK
LD 4482.07  ; PAIR POLE NG
OR 4484.07  ; NEXT POLE NG
AND ALL_OK
ORLD
AND H146.15  ; IMPULSE_STEP 15
MOV(021) #1 E2810  ; IMPULSE MEASUREMENT JUDGMENT RESULT (1:OK,2:NG)
AND<>(305) E2819 #2  ; Synthesis OK
MOV(021) #1 E2819  ; Synthesis OK
; rung 94
LD 4482.07  ; PAIR POLE NG
OR 4484.07  ; NEXT POLE NG
ANDNOT ALL_OK
AND H146.15  ; IMPULSE_STEP 15
MOV(021) #2 E2810  ; IMPULSE MEASUREMENT JUDGMENT RESULT (1:OK,2:NG)
MOV(021) #2 E2819  ; Synthesis OK
; rung 95
LD H146.15  ; IMPULSE_STEP 15
OUT TR0
LD 4484.09  ; NEXT POLE  OK
LD ALL_OK
AND 4484.07  ; NEXT POLE NG
ORLD
ANDLD
MOV(021) #1 E2812  ; IMPULSE NEXT POLE JUDGMENT RESULT (1:OK,2:NG)
LD TR0
AND 4484.07  ; NEXT POLE NG
ANDNOT ALL_OK
MOV(021) #2 E2812  ; IMPULSE NEXT POLE JUDGMENT RESULT (1:OK,2:NG)

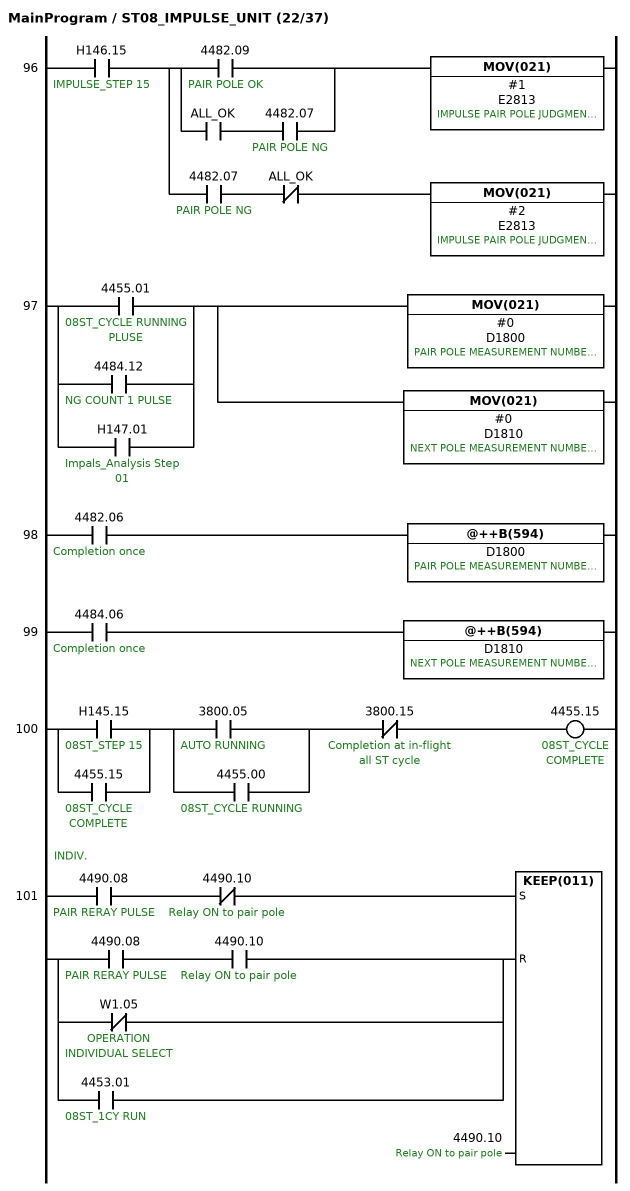
; rung 96
LD H146.15  ; IMPULSE_STEP 15
OUT TR0
LD 4482.09  ; PAIR POLE OK
LD ALL_OK
AND 4482.07  ; PAIR POLE NG
ORLD
ANDLD
MOV(021) #1 E2813  ; IMPULSE PAIR POLE JUDGMENT RESULT (1:OK,2:NG)
LD TR0
AND 4482.07  ; PAIR POLE NG
ANDNOT ALL_OK
MOV(021) #2 E2813  ; IMPULSE PAIR POLE JUDGMENT RESULT (1:OK,2:NG)
; rung 97
LD 4455.01  ; 08ST_CYCLE RUNNING PLUSE
OR 4484.12  ; NG COUNT 1 PULSE
OR H147.01  ; Impals_Analysis Step 01
MOV(021) #0 D1800  ; PAIR POLE MEASUREMENT NUMBER OF TIMES
MOV(021) #0 D1810  ; NEXT POLE MEASUREMENT NUMBER OF TIMES
; rung 98
LD 4482.06  ; Completion once
@++B(594) D1800  ; PAIR POLE MEASUREMENT NUMBER OF TIMES
; rung 99
LD 4484.06  ; Completion once
@++B(594) D1810  ; NEXT POLE MEASUREMENT NUMBER OF TIMES
; rung 100
LD H145.15  ; 08ST_STEP 15
OR 4455.15  ; 08ST_CYCLE COMPLETE
LD 3800.05  ; AUTO RUNNING
OR 4455.00  ; 08ST_CYCLE RUNNING
ANDLD
ANDNOT 3800.15  ; Completion at in-flight all ST cycle
OUT 4455.15  ; 08ST_CYCLE COMPLETE
; rung 101: INDIV.
LD 4490.08  ; PAIR RERAY PULSE
ANDNOT 4490.10  ; Relay ON to pair pole
LD 4490.08  ; PAIR RERAY PULSE
AND 4490.10  ; Relay ON to pair pole
ORNOT W1.05  ; OPERATION INDIVIDUAL SELECT
OR 4453.01  ; 08ST_1CY RUN
KEEP(011) 4490.10  ; Relay ON to pair pole

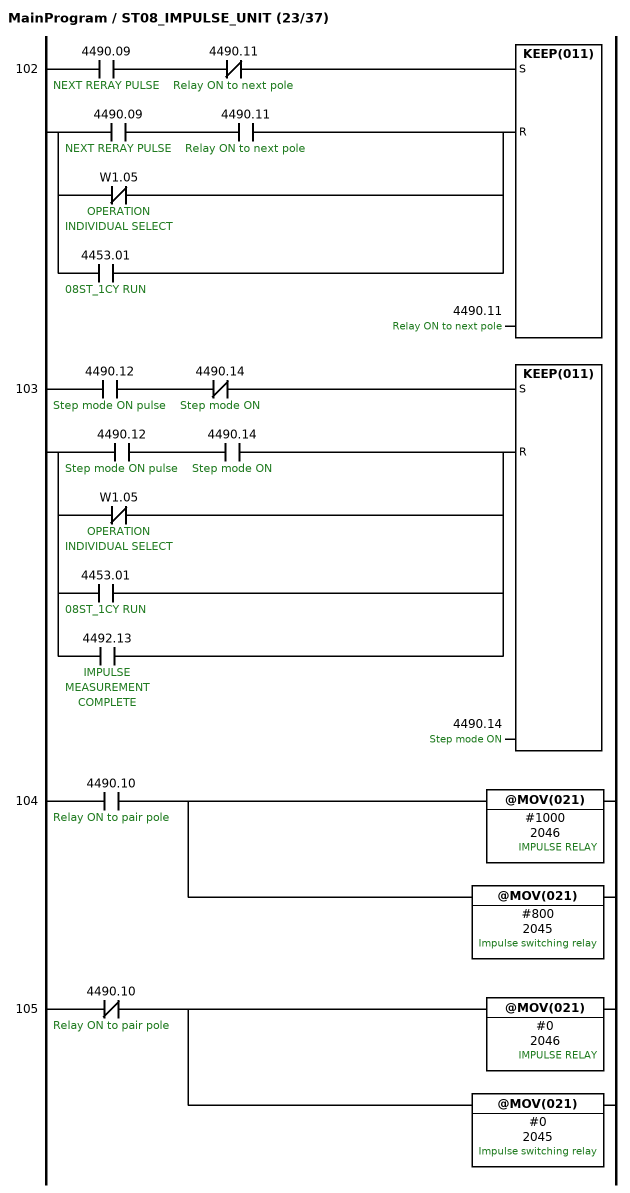
; rung 102
LD 4490.09  ; NEXT RERAY PULSE
ANDNOT 4490.11  ; Relay ON to next pole
LD 4490.09  ; NEXT RERAY PULSE
AND 4490.11  ; Relay ON to next pole
ORNOT W1.05  ; OPERATION INDIVIDUAL SELECT
OR 4453.01  ; 08ST_1CY RUN
KEEP(011) 4490.11  ; Relay ON to next pole
; rung 103
LD 4490.12  ; Step mode ON pulse
ANDNOT 4490.14  ; Step mode ON
LD 4490.12  ; Step mode ON pulse
AND 4490.14  ; Step mode ON
ORNOT W1.05  ; OPERATION INDIVIDUAL SELECT
OR 4453.01  ; 08ST_1CY RUN
OR 4492.13  ; IMPULSE MEASUREMENT COMPLETE
KEEP(011) 4490.14  ; Step mode ON
; rung 104
LD 4490.10  ; Relay ON to pair pole
@MOV(021) #1000 2046  ; IMPULSE RELAY
@MOV(021) #800 2045  ; Impulse switching relay
; rung 105
LDNOT 4490.10  ; Relay ON to pair pole
@MOV(021) #0 2046  ; IMPULSE RELAY
@MOV(021) #0 2045  ; Impulse switching relay

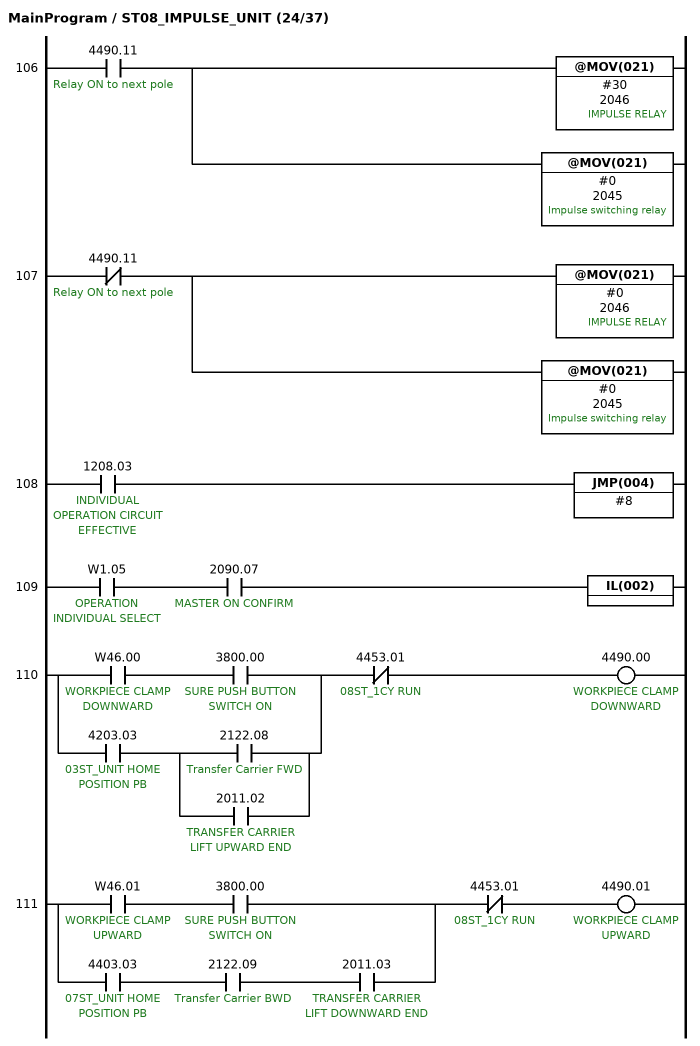
; rung 106
LD 4490.11  ; Relay ON to next pole
@MOV(021) #30 2046  ; IMPULSE RELAY
@MOV(021) #0 2045  ; Impulse switching relay
; rung 107
LDNOT 4490.11  ; Relay ON to next pole
@MOV(021) #0 2046  ; IMPULSE RELAY
@MOV(021) #0 2045  ; Impulse switching relay
; rung 108
LD 1208.03  ; INDIVIDUAL OPERATION CIRCUIT EFFECTIVE
JMP(004) #8
; rung 109
LD W1.05  ; OPERATION INDIVIDUAL SELECT
AND 2090.07  ; MASTER ON CONFIRM
IL(002)
; rung 110
LD W46.00  ; WORKPIECE CLAMP DOWNWARD
AND 3800.00  ; SURE PUSH BUTTON SWITCH ON
LD 4203.03  ; 03ST_UNIT HOME POSITION PB
LD 2122.08  ; Transfer Carrier FWD
OR 2011.02  ; TRANSFER CARRIER LIFT UPWARD END
ANDLD
ORLD
ANDNOT 4453.01  ; 08ST_1CY RUN
OUT 4490.00  ; WORKPIECE CLAMP DOWNWARD
; rung 111
LD W46.01  ; WORKPIECE CLAMP UPWARD
AND 3800.00  ; SURE PUSH BUTTON SWITCH ON
LD 4403.03  ; 07ST_UNIT HOME POSITION PB
AND 2122.09  ; Transfer Carrier BWD
AND 2011.03  ; TRANSFER CARRIER LIFT DOWNWARD END
ORLD
ANDNOT 4453.01  ; 08ST_1CY RUN
OUT 4490.01  ; WORKPIECE CLAMP UPWARD

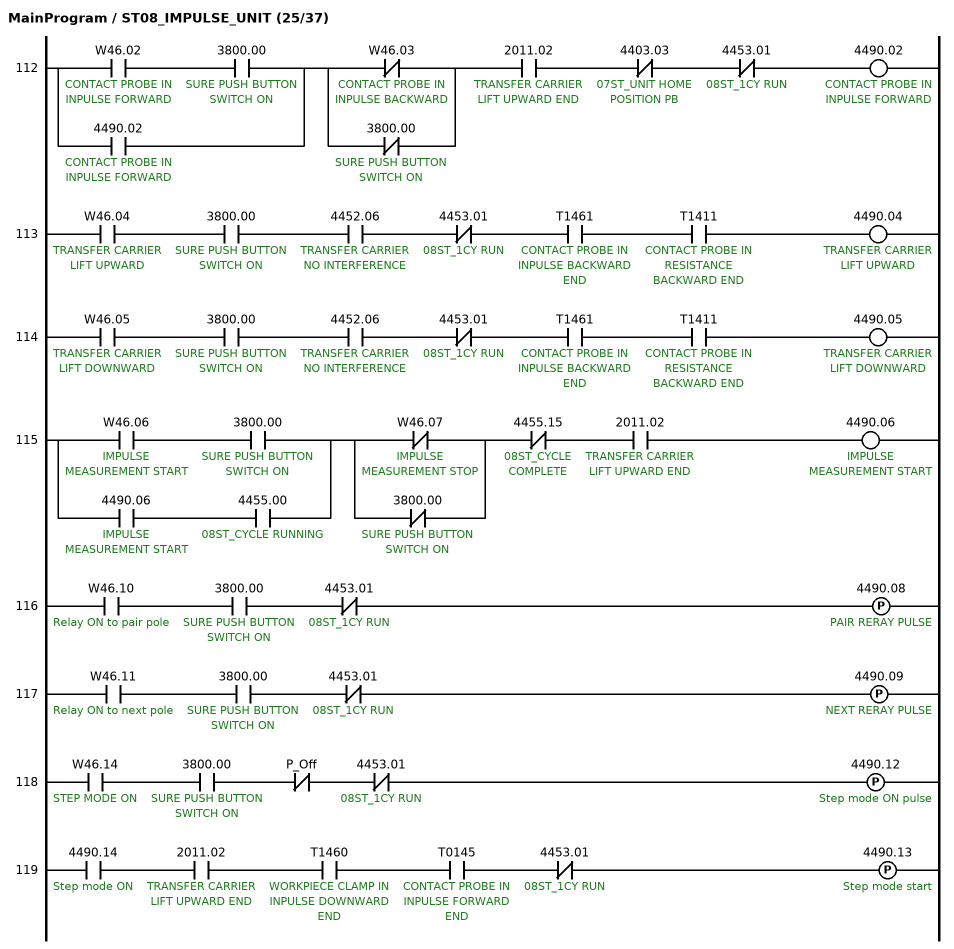
; rung 112
LD W46.02  ; CONTACT PROBE IN INPULSE FORWARD
AND 3800.00  ; SURE PUSH BUTTON SWITCH ON
OR 4490.02  ; CONTACT PROBE IN INPULSE FORWARD
LDNOT W46.03  ; CONTACT PROBE IN INPULSE BACKWARD
ORNOT 3800.00  ; SURE PUSH BUTTON SWITCH ON
ANDLD
AND 2011.02  ; TRANSFER CARRIER LIFT UPWARD END
ANDNOT 4403.03  ; 07ST_UNIT HOME POSITION PB
ANDNOT 4453.01  ; 08ST_1CY RUN
OUT 4490.02  ; CONTACT PROBE IN INPULSE FORWARD
; rung 113
LD W46.04  ; TRANSFER CARRIER LIFT UPWARD
AND 3800.00  ; SURE PUSH BUTTON SWITCH ON
AND 4452.06  ; TRANSFER CARRIER NO INTERFERENCE
ANDNOT 4453.01  ; 08ST_1CY RUN
AND T1461  ; CONTACT PROBE IN INPULSE BACKWARD END
AND T1411  ; CONTACT PROBE IN RESISTANCE BACKWARD END
OUT 4490.04  ; TRANSFER CARRIER LIFT UPWARD
; rung 114
LD W46.05  ; TRANSFER CARRIER LIFT DOWNWARD
AND 3800.00  ; SURE PUSH BUTTON SWITCH ON
AND 4452.06  ; TRANSFER CARRIER NO INTERFERENCE
ANDNOT 4453.01  ; 08ST_1CY RUN
AND T1461  ; CONTACT PROBE IN INPULSE BACKWARD END
AND T1411  ; CONTACT PROBE IN RESISTANCE BACKWARD END
OUT 4490.05  ; TRANSFER CARRIER LIFT DOWNWARD
; rung 115
LD W46.06  ; IMPULSE MEASUREMENT START
AND 3800.00  ; SURE PUSH BUTTON SWITCH ON
LD 4490.06  ; IMPULSE MEASUREMENT START
AND 4455.00  ; 08ST_CYCLE RUNNING
ORLD
LDNOT W46.07  ; IMPULSE MEASUREMENT STOP
ORNOT 3800.00  ; SURE PUSH BUTTON SWITCH ON
ANDLD
ANDNOT 4455.15  ; 08ST_CYCLE COMPLETE
AND 2011.02  ; TRANSFER CARRIER LIFT UPWARD END
OUT 4490.06  ; IMPULSE MEASUREMENT START
; rung 116
LD W46.10  ; Relay ON to pair pole
AND 3800.00  ; SURE PUSH BUTTON SWITCH ON
ANDNOT 4453.01  ; 08ST_1CY RUN
DIFU(013) 4490.08  ; PAIR RERAY PULSE
; rung 117
LD W46.11  ; Relay ON to next pole
AND 3800.00  ; SURE PUSH BUTTON SWITCH ON
ANDNOT 4453.01  ; 08ST_1CY RUN
DIFU(013) 4490.09  ; NEXT RERAY PULSE
; rung 118
LD W46.14  ; STEP MODE ON
AND 3800.00  ; SURE PUSH BUTTON SWITCH ON
ANDNOT P_Off
ANDNOT 4453.01  ; 08ST_1CY RUN
DIFU(013) 4490.12  ; Step mode ON pulse
; rung 119
LD 4490.14  ; Step mode ON
AND 2011.02  ; TRANSFER CARRIER LIFT UPWARD END
AND T1460  ; WORKPIECE CLAMP IN INPULSE DOWNWARD END
AND T0145  ; CONTACT PROBE IN INPULSE FORWARD END
ANDNOT 4453.01  ; 08ST_1CY RUN
DIFU(013) 4490.13  ; Step mode start

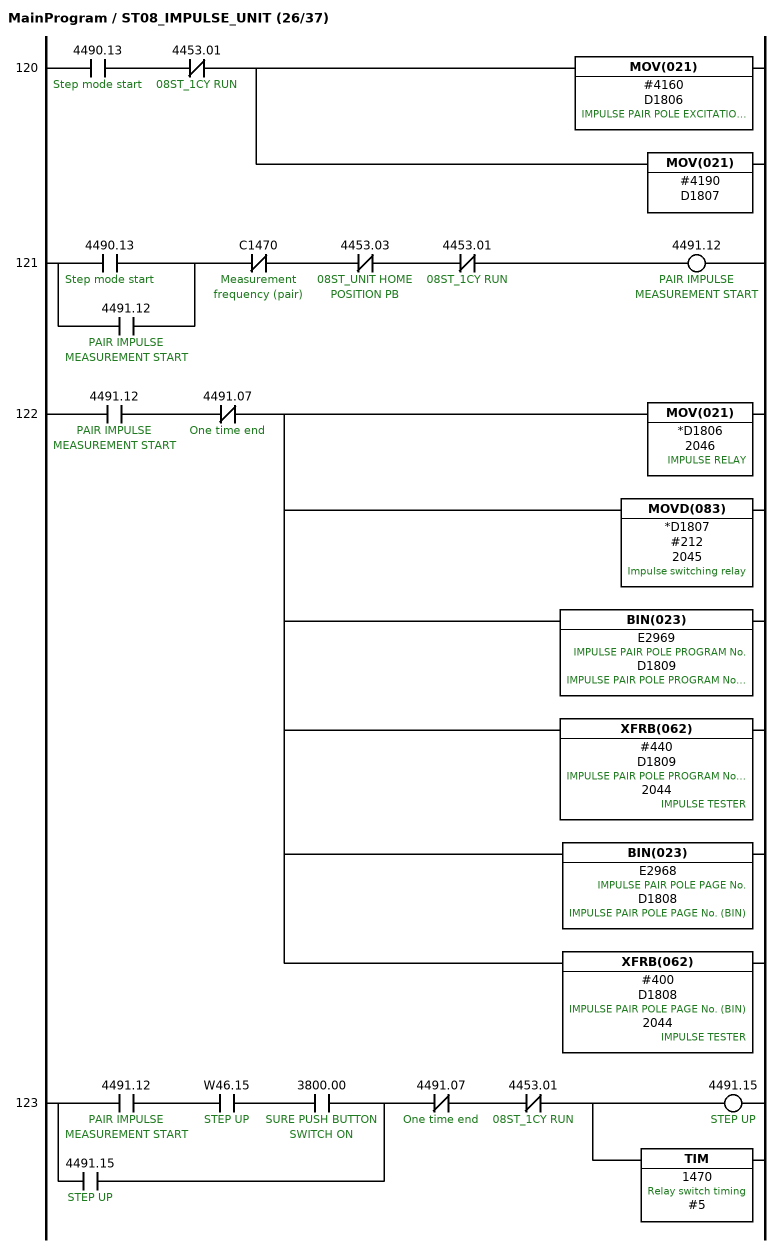
; rung 120
LD 4490.13  ; Step mode start
ANDNOT 4453.01  ; 08ST_1CY RUN
MOV(021) #4160 D1806  ; IMPULSE PAIR POLE EXCITATION PATTERN DM STORING(INDIVIDUAL)
MOV(021) #4190 D1807
; rung 121
LD 4490.13  ; Step mode start
OR 4491.12  ; PAIR IMPULSE MEASUREMENT START
ANDNOT C1470  ; Measurement frequency (pair)
ANDNOT 4453.03  ; 08ST_UNIT HOME POSITION PB
ANDNOT 4453.01  ; 08ST_1CY RUN
OUT 4491.12  ; PAIR IMPULSE MEASUREMENT START
; rung 122
LD 4491.12  ; PAIR IMPULSE MEASUREMENT START
ANDNOT 4491.07  ; One time end
MOV(021) *D1806 2046  ; IMPULSE RELAY
MOVD(083) *D1807 #212 2045  ; Impulse switching relay
BIN(023) E2969 D1809  ; IMPULSE PAIR POLE PROGRAM No., IMPULSE PAIR POLE PROGRAM No. (BIN)
XFRB(062) #440 D1809 2044  ; IMPULSE PAIR POLE PROGRAM No. (BIN), IMPULSE TESTER
BIN(023) E2968 D1808  ; IMPULSE PAIR POLE PAGE No., IMPULSE PAIR POLE PAGE No. (BIN)
XFRB(062) #400 D1808 2044  ; IMPULSE PAIR POLE PAGE No. (BIN), IMPULSE TESTER
; rung 123
LD 4491.12  ; PAIR IMPULSE MEASUREMENT START
AND W46.15  ; STEP UP
AND 3800.00  ; SURE PUSH BUTTON SWITCH ON
OR 4491.15  ; STEP UP
ANDNOT 4491.07  ; One time end
ANDNOT 4453.01  ; 08ST_1CY RUN
OUT 4491.15  ; STEP UP
TIM 1470 #5  ; Relay switch timing

